(* Whether the bridge itself is established; local/remote operational state and device presence, before any data-quality signal is meaningful. *)
TYPE E_BridgeLinkStatus :
(
    Connected,                    // local State = OP, far device present, far side TxPDOState = 0 (OP)
    LocalNotOperational,          // local State <> OP
    ExternalDeviceNotConnected,   // far device not present
    RemoteNotOperational          // far device present but TxPDOState <> 0
) UDINT;
END_TYPE

(* stored: Version 1.1.0.1
   DUT E_BridgeLinkStatus: Id {c3a7e156-8d24-4f91-a06b-1e3d9c5a2f78} *)
